Universal Robots PolyScope program: Arla0.2.urp

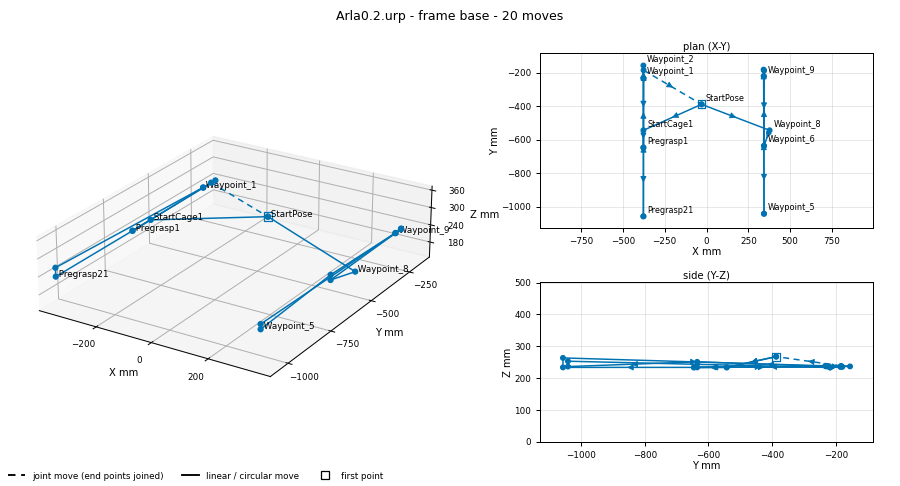
[picture p0: tool path of Arla0.2.urp in frame base, 20 of 20 moves have a stored position in this frame; points joined in program order, loops and branches not executed]
Program Arla0.2 (installation=default directory=/programs/usbdisk createdIn=5.11.4.108353 lastSavedIn=5.9.1.1031110 robotSerialNumber=20185000125)
Calibrated DH parameters: a=[0.000009, -0.582937, -0.560313, -0.000136, -0.000015, 0]; d=[0.181003, 62.966139, -25.546705, -37.245036, 0.119984, 0.115761]; alpha=[1.570753, -0.002987, -0.002977, 1.572291, -1.570292, 0]; deltaTheta=[-0.000001, -0.312112, 0.115839, 0.196276, -0.000002, 0]
Robot Program (runOnlyOnce=true)
  Folder ResetForce
    Wait Condition expression=is_steady()
    Wait Sleep waitTime=0.25
    Script: zero_ftsensor()
    Wait Sleep waitTime=0.25
  Timer (action=Start) variable(name=timer_1)
  MoveJ speed 30 deg/s, acceleration 40 deg/s^2 (useActiveTCP=true) feature=Base
    Waypoint StartPose: motionParameters(jointSpeed=0.523599 jointAcceleration=0.698132 cartesianSpeed=0.25 cartesianAcceleration=1.2); TCP in base x=-29.649 y=-387.378 z=267.725 mm, rx=0 ry=-3.1416 rz=0 rad; joints [-67.884, -70.586, -150.404, -49.041, 89.902, 22.237] deg
  Folder Cage1
    MoveL speed 250 mm/s, acceleration 1200 mm/s^2 (useActiveTCP=true) feature=Base
      Waypoint StartCage1: TCP in base x=-377.018 y=-542.594 z=233.918 mm, rx=-0.1647 ry=-3.1372 rz=0.0003 rad; joints [-109.613, -103.066, -125.349, -41.605, 89.828, -13.516] deg
    MoveL speed 250 mm/s, acceleration 1200 mm/s^2 (useActiveTCP=true) feature=Base
      Waypoint Pregrasp1: TCP in base x=-377.023 y=-645.691 z=233.925 mm, rx=0.1472 ry=3.1381 rz=-0.0004 rad; joints [-106.906, -109.721, -115.734, -44.56, 89.809, -11.457] deg
    Force Frame feature=Base; selection=[0, 0, 1, 0, 0, 0]; wrench=[0, 10, 225, 0, 0, 0]; limitsForce=[0.15, 0.15, 0.15, 1.047198, 1.047198, 1.047198]; limitsMotion=[0.1, 0.1, 0.1, 0.349066, 0.349066, 0.349066]
      Set DigitalOutput pin=digital_out[0]; digitalValue=1
      Wait Sleep waitTime=0.5
    MoveL speed 100 mm/s, acceleration 1200 mm/s^2 (useActiveTCP=true) feature=Base
      MoveDirectionNode (selectedDirection=YPlus)
        Until DISTANCE (allowActions=false deceleration=3 distanceNodeType=STOP) Distance=0.1; motionParameters(blendRadius=0)
    Set DigitalOutput pin=digital_out[0]; digitalValue=0
    MoveL speed 250 mm/s, acceleration 1200 mm/s^2 (useActiveTCP=true) feature=Base
      MoveDirectionNode (selectedDirection=YPlus)
        Until DISTANCE (allowActions=false deceleration=3 distanceNodeType=STOP) Distance=0.315; motionParameters(blendRadius=0)
    MoveL speed 250 mm/s, acceleration 1200 mm/s^2 (useActiveTCP=true) feature=Base
      Waypoint Waypoint_1: TCP in base x=-377.05 y=-230.69 z=236.965 mm, rx=-0.1473 ry=-3.1381 rz=-0.0006 rad; joints [-125.334, -81.964, -147.416, -40.639, 89.988, -29.959] deg; TCP offset x=0 y=0 z=0 mm, rx=0 ry=0 rz=0 rad
    MoveL speed 250 mm/s, acceleration 1200 mm/s^2 (useActiveTCP=true) feature=Base
      Waypoint Waypoint_2: TCP in base x=-377.05 y=-155.463 z=236.965 mm, rx=-0.1473 ry=-3.1381 rz=-0.0006 rad; joints [-132.311, -77.472, -150.605, -41.939, 89.986, -36.936] deg
    Wait Sleep waitTime=2
    MoveL speed 250 mm/s, acceleration 1200 mm/s^2 (useActiveTCP=true) feature=Base
      Waypoint Pregrasp1: TCP in base x=-377.023 y=-645.691 z=233.925 mm, rx=0.1472 ry=3.1381 rz=-0.0004 rad; joints [-106.906, -109.721, -115.734, -44.56, 89.809, -11.457] deg
    MoveL speed 250 mm/s, acceleration 1200 mm/s^2 (useActiveTCP=true) feature=Base
      MoveDirectionNode (selectedDirection=ZPlus)
        Until DISTANCE (allowActions=false deceleration=3 distanceNodeType=STOP) Distance=0.007; motionParameters(blendRadius=0)
    MoveL speed 250 mm/s, acceleration 1200 mm/s^2 (useActiveTCP=true) feature=Base
      Waypoint Pregrasp21: TCP in base x=-377.061 y=-1056.7 z=233.886 mm, rx=-0.1648 ry=-3.1372 rz=0.0002 rad; joints [-100.743, -139.405, -64.21, -66.406, 89.701, -4.674] deg
    MoveL speed 300 mm/s, acceleration 1200 mm/s^2 (useActiveTCP=true) feature=Base
      Waypoint Pregrasp22: TCP in base x=-377.043 y=-1056.692 z=263.615 mm, rx=-0.1648 ry=-3.1372 rz=0.0001 rad; joints [-100.742, -138.214, -63.213, -68.601, 89.701, -4.664] deg
    MoveL speed 250 mm/s, acceleration 1200 mm/s^2 (useActiveTCP=true) feature=Base
      MoveDirectionNode (selectedDirection=YPlus)
        Until DISTANCE (allowActions=false deceleration=3 distanceNodeType=STOP) Distance=0.405; motionParameters(blendRadius=0)
    Force Frame feature=Base; selection=[0, 0, 1, 0, 0, 0]; wrench=[0, 10, 225, 0, 0, 0]; limitsForce=[0.15, 0.15, 0.15, 1.047198, 1.047198, 1.047198]; limitsMotion=[0.1, 0.1, 0.1, 0.349066, 0.349066, 0.349066]
      Wait Sleep waitTime=0.7
    MoveL speed 100 mm/s, acceleration 1200 mm/s^2 (useActiveTCP=true) feature=Base
      MoveDirectionNode (selectedDirection=YPlus)
        Until DISTANCE (allowActions=false deceleration=3 distanceNodeType=STOP) Distance=0.415; motionParameters(blendRadius=0)
    MoveL speed 300 mm/s, acceleration 1200 mm/s^2 (useActiveTCP=true) feature=Base
      Waypoint Waypoint_3: TCP in base x=-375.947 y=-233.163 z=238.766 mm, rx=0.1646 ry=3.1354 rz=0.0122 rad; joints [-125.091, -81.854, -147.182, -41.428, 89.742, -28.973] deg
    MoveL speed 300 mm/s, acceleration 1200 mm/s^2 (useActiveTCP=true) feature=Base
      Waypoint Waypoint_4: TCP in base x=-375.933 y=-183.47 z=238.741 mm, rx=0.1647 ry=3.1353 rz=0.0123 rad; joints [-129.455, -78.758, -149.443, -42.254, 89.717, -33.331] deg
    Wait Sleep waitTime=2
  MoveJ speed 30 deg/s, acceleration 40 deg/s^2 (useActiveTCP=true) feature=Base
    Waypoint StartPose: motionParameters(jointSpeed=0.523599 jointAcceleration=0.698132 cartesianSpeed=0.25 cartesianAcceleration=1.2); TCP in base x=-29.649 y=-387.378 z=267.725 mm, rx=0 ry=-3.1416 rz=0 rad; joints [-67.884, -70.586, -150.404, -49.041, 89.902, 22.237] deg
  Timer (action=Start) variable=timer_1
  Folder Cage2
    MoveL speed 400 mm/s, acceleration 1200 mm/s^2 (useActiveTCP=true) feature=Base
      Waypoint Waypoint_8: TCP in base x=377.02 y=-542.594 z=233.918 mm, rx=-0.1647 ry=-3.1372 rz=0.0003 rad; joints [-40.025, -103.065, -125.347, -41.613, 89.819, 56.073] deg; TCP offset x=0 y=0 z=0 mm, rx=0 ry=0 rz=0 rad
    MoveL speed 400 mm/s, acceleration 1200 mm/s^2 (useActiveTCP=true) feature=Base
      Waypoint Waypoint_6: TCP in base x=343.499 y=-635.479 z=233.957 mm, rx=-0.1647 ry=-3.1373 rz=0.0004 rad; joints [-47.751, -107.813, -118.586, -43.62, 89.801, 48.338] deg
    Set DigitalOutput pin=digital_out[0]; digitalValue=1
    var_1 := get_actual_tcp_pose()
    Force Frame feature=Base; selection=[0, 0, 1, 0, 0, 0]; wrench=[0, 10, 225, 0, 0, 0]; limitsForce=[0.15, 0.15, 0.15, 1.047198, 1.047198, 1.047198]; limitsMotion=[0.1, 0.1, 0.1, 0.349066, 0.349066, 0.349066]
      Loop While (checkContinuously=false) expression=var_1[2] < 0.275
        var_1 := get_actual_tcp_pose()
    var_1 := get_actual_tcp_pose()
    Force Frame feature=Base; selection=[0, 0, 1, 0, 0, 0]; wrench=[0, 10, 225, 0, 0, 0]; limitsForce=[0.15, 0.15, 0.15, 1.047198, 1.047198, 1.047198]; limitsMotion=[0.1, 0.1, 0.1, 0.349066, 0.349066, 0.349066]
      Set DigitalOutput pin=digital_out[0]; digitalValue=1
    MoveL speed 250 mm/s, acceleration 1200 mm/s^2 (useActiveTCP=true) feature=Base
      MoveDirectionNode (selectedDirection=YPlus)
        Until DISTANCE (allowActions=false deceleration=3 distanceNodeType=STOP) Distance=0.1; motionParameters(blendRadius=0)
    Set DigitalOutput pin=digital_out[0]; digitalValue=0
    MoveL speed 250 mm/s, acceleration 1200 mm/s^2 (useActiveTCP=true) feature=Base
      MoveDirectionNode (selectedDirection=YPlus)
        Until DISTANCE (allowActions=false deceleration=3 distanceNodeType=STOP) Distance=0.315; motionParameters(blendRadius=0)
    MoveL speed 400 mm/s, acceleration 1200 mm/s^2 (useActiveTCP=true) feature=Base
      Waypoint Waypoint_9: TCP in base x=343.344 y=-220.193 z=235.398 mm, rx=-0.1642 ry=-3.1366 rz=-0.0011 rad; joints [-7.535, -77.835, -150.69, -41.549, 89.937, 88.568] deg
    MoveL speed 400 mm/s, acceleration 1200 mm/s^2 (useActiveTCP=true) feature=Base
      Waypoint Waypoint_10: TCP in base x=343.967 y=-185.915 z=235.406 mm, rx=-0.1641 ry=-3.1366 rz=-0.0011 rad; joints [-2.083, -75.381, -152.234, -42.453, 89.944, 94.019] deg
    Halt
    MoveL speed 400 mm/s, acceleration 1200 mm/s^2 (useActiveTCP=true) feature=Base
      Waypoint Waypoint_11: TCP in base x=343.517 y=-635.445 z=251.337 mm, rx=-0.1646 ry=-3.1372 rz=0.0002 rad; joints [-47.75, -106.495, -118.012, -45.518, 89.802, 48.342] deg
    MoveL speed 400 mm/s, acceleration 1200 mm/s^2 (useActiveTCP=true) feature=Base
      Waypoint Waypoint_5: TCP in base x=343.551 y=-1041.016 z=236.521 mm, rx=-0.1645 ry=-3.1372 rz=0.0001 rad; joints [-62.635, -136.879, -68.665, -64.484, 89.703, 33.424] deg
    MoveL speed 400 mm/s, acceleration 1200 mm/s^2 (useActiveTCP=true) feature=Base
      Waypoint Waypoint_7: TCP in base x=343.552 y=-1041.014 z=253.298 mm, rx=-0.1644 ry=-3.1372 rz=0.0001 rad; joints [-62.635, -136.166, -68.133, -65.731, 89.702, 33.426] deg
    MoveL speed 400 mm/s, acceleration 1200 mm/s^2 (useActiveTCP=true) feature=Base
      MoveDirectionNode (selectedDirection=YPlus)
        Until DISTANCE (allowActions=false deceleration=3 distanceNodeType=STOP) Distance=0.405; motionParameters(blendRadius=0)
    var_1 := get_actual_tcp_pose()
    Force Frame feature=Base; selection=[0, 0, 1, 0, 0, 0]; wrench=[0, 10, 225, 0, 0, 0]; limitsForce=[0.15, 0.15, 0.15, 1.047198, 1.047198, 1.047198]; limitsMotion=[0.1, 0.1, 0.1, 0.349066, 0.349066, 0.349066]
      Loop While (checkContinuously=false) expression=var_1[2] < 0.275
        var_1 := get_actual_tcp_pose()
    Wait Sleep waitTime=0.5
    MoveL speed 200 mm/s, acceleration 400 mm/s^2 (useActiveTCP=true) feature=Base
      MoveDirectionNode (selectedDirection=YPlus)
        Until DISTANCE (allowActions=false deceleration=3 distanceNodeType=STOP) Distance=0.415; motionParameters(blendRadius=0.05)
    MoveL speed 400 mm/s, acceleration 1200 mm/s^2 (useActiveTCP=true) feature=Base
      Waypoint Waypoint_12: TCP in base x=341.332 y=-218.663 z=233.476 mm, rx=-0.1641 ry=-3.132 rz=-0.007 rad; joints [-7.4, -77.77, -150.937, -41.641, 90.132, 88.707] deg
    MoveL speed 400 mm/s, acceleration 1200 mm/s^2 (useActiveTCP=true) feature=Base
      Waypoint Waypoint_13: TCP in base x=341.336 y=-179.93 z=235.41 mm, rx=-0.164 ry=-3.132 rz=-0.007 rad; joints [-1.184, -74.618, -152.606, -43.097, 90.172, 94.922] deg
  Timer (action=Stop) variable=timer_1
